Yaskawa INFORM job: KRIS6(-12_90).JBI

/JOB
//NAME KRIS6(-12_90)
//POS
///NPOS 178,178,178,10,0,0
///TOOL 0
///POSTYPE PULSE
///PULSE
C00000=-6764,-164331,-134999,2181,78960,314
C00001=-119255,-47763,-118129,2201,84733,937
C00002=-119348,-33730,-112223,2255,86453,948
C00003=-119057,-93541,-129160,2121,87990,859
C00004=-118979,-101393,-133254,2097,92873,863
C00005=-119932,-77312,-125419,2251,104410,725
C00006=-119932,-79807,-125118,2239,102944,696
C00007=-119932,-78534,-125283,2248,103699,711
C00008=-119946,-74107,-123441,2264,104839,725
C00009=-119932,-78534,-125283,2248,103699,711
C00010=-119867,-91458,-132961,2208,101782,695
C00011=-119929,-73545,-130238,2283,96557,768
C00012=-119929,-73545,-130238,2283,96557,768
C00013=-119957,-58817,-118616,2436,108946,925
C00014=-123171,-49481,-113469,3470,112784,170
C00015=-123153,-49145,-112726,3457,112499,166
C00016=-123153,-51096,-112549,3427,111389,133
C00017=-123153,-49599,-112689,3450,112241,159
C00018=-123109,-46536,-111045,3454,112801,187
C00019=-123280,-52221,-117750,3539,114010,179
C00020=-123574,-64329,-127676,3623,101325,100
C00021=-123574,-64329,-127676,3623,101325,100
C00022=-123766,-59413,-122861,3666,112999,36
C00023=-125942,-52580,-116093,4293,112422,-554
C00024=-126600,-50426,-113316,4465,111850,-748
C00025=-126600,-52772,-113093,4419,110512,-799
C00026=-126600,-51256,-113243,4448,111381,-766
C00027=-126484,-47796,-111410,4439,112022,-709
C00028=-126600,-51256,-113243,4448,111381,-766
C00029=-127517,-71417,-126819,4648,109419,-1089
C00030=-127517,-71417,-126819,4648,95207,-1089
C00031=-127517,-71417,-126819,4648,95207,-1089
C00032=-127517,-73529,-126819,4648,106019,-1089
C00033=-127727,-61749,-119091,4751,107320,-1094
C00034=-130093,-58052,-115859,5494,107341,-1725
C00035=-130093,-60399,-115576,5448,105965,-1787
C00036=-130093,-58676,-115790,5482,106977,-1740
C00037=-129907,-55107,-114011,5451,107705,-1657
C00038=-130162,-58740,-116586,5519,107435,-1737
C00039=-131204,-71916,-126481,5822,106811,-2045
C00040=-131204,-71916,-126481,5822,93687,-2045
C00041=-131204,-71916,-126481,5822,93687,-2045
C00042=-131204,-71916,-126481,5822,105723,-2045
C00043=-130617,-65357,-120996,5631,105686,-1890
C00044=-134640,-60773,-116482,6918,105500,-2981
C00045=-134640,-62624,-116236,6876,104404,-3044
C00046=-134640,-61323,-116413,6905,105177,-2999
C00047=-134343,-57381,-114492,6841,105996,-2874
C00048=-134640,-61323,-116413,6905,105177,-2999
C00049=-133458,-71885,-125928,6541,105529,-2666
C00050=-133867,-78779,-128765,6711,91394,-2865
C00051=-133867,-78779,-128765,6711,91394,-2865
C00052=-133867,-78779,-128765,6711,103158,-2865
C00053=-137702,-64049,-118295,8003,104543,-3826
C00054=-138377,-60786,-116211,8241,104986,-3979
C00055=-138377,-63432,-115832,8173,103411,-4088
C00056=-138377,-61523,-116113,8222,104554,-4010
C00057=-138001,-57618,-114209,8136,105352,-3854
C00058=-138804,-63923,-118462,8370,104797,-4109
C00059=-114789,-54631,-113943,-15836,109322,15159
C00060=-117446,-46661,-107682,-17796,110513,16745
C00061=-135138,-47810,-110215,2755,110872,-639
C00062=-122706,-51038,-111939,2830,110281,-732
C00063=-104898,-47309,-109719,-2181,110784,3733
C00064=-113247,-41947,-106722,9396,112942,-6495
C00065=-115201,-45518,-111139,10036,113978,-6928
C00066=-109888,-67792,-124928,-2208,109623,3796
C00067=-109888,-67792,-124928,-2208,92487,3796
C00068=-109888,-67792,-124928,-2208,92487,3796
C00069=-109888,-67792,-124928,-2208,107991,3796
C00070=-119439,-51982,-113666,11445,111008,-7659
C00071=-117726,-48338,-109777,10887,110325,-7260
C00072=-100866,-50921,-111009,-8782,109155,9371
C00073=-117735,-56763,-114072,-3538,107088,4956
C00074=-137822,-52486,-111893,2748,107867,-389
C00075=-124279,-42666,-106545,-13838,112284,13520
C00076=-119511,-49264,-112664,-15270,113256,14701
C00077=-119402,-57305,-120939,-15547,101345,14582
C00078=-119402,-57305,-120939,-15547,101345,14582
C00079=-119402,-57305,-120939,-15547,109505,14582
C00080=-122292,-51504,-112613,-14389,109095,14125
C00081=-124558,-45323,-107894,-13672,111001,13362
C00082=-143884,-51554,-111193,8957,108316,-5281
C00083=-133478,-57417,-114087,5875,106433,-2802
C00084=-120249,-59696,-115195,2556,105532,-22
C00085=-132290,-46931,-108595,16593,111984,-11759
C00086=-136159,-47694,-113124,18059,114858,-12388
C00087=-139576,-57528,-118771,18775,113901,-13510
C00088=-140360,-69519,-123680,18885,96024,-14170
C00089=-140360,-69519,-123678,18885,96029,-14170
C00090=-141278,-80916,-127529,19144,105606,-14918
C00091=-135966,-58193,-116482,18148,109309,-12780
C00092=-133070,-49776,-109673,17224,110272,-12037
C00093=-115680,-63515,-116432,-2666,103196,4100
C00094=-124283,-63101,-116291,-1790,103261,3381
C00095=-141256,-57210,-113499,5768,104997,-2724
C00096=-125849,-50663,-110250,-12105,107953,11564
C00097=-122691,-57409,-116127,-13110,108460,12368
C00098=-121144,-64717,-120648,-13506,107699,12878
C00099=-121162,-72749,-124196,-13450,93226,13080
C00100=-121162,-72749,-124196,-13450,93226,13080
C00101=-121162,-72749,-124196,-13450,105330,13080
C00102=-121331,-50205,-111480,-16610,110216,14952
C00103=-123990,-47823,-108385,-15715,109173,14365
C00104=-142128,-42054,-107579,5566,113340,-3269
C00105=-131359,-47053,-110363,2420,112110,-462
C00106=-117986,-48725,-111182,-1462,111698,3083
C00107=-133863,-43680,-107086,16750,113488,-14506
C00108=-140868,-51734,-116509,18965,116153,-16042
C00109=-142662,-63919,-124161,19179,114978,-16761
C00110=-142662,-63919,-124161,19179,98114,-16761
C00111=-142662,-63919,-124161,19179,98114,-16761
C00112=-145044,-62011,-123293,19965,112812,-17284
C00113=-140059,-55739,-114817,18192,110093,-16328
C00114=-137449,-52455,-110379,17263,108669,-15828
C00115=-120073,-53031,-112853,-3294,109306,530
C00116=-131848,-51289,-111914,267,109461,-2602
C00117=-144044,-45121,-108584,3992,110813,-5796
C00118=-132169,-40707,-106079,-10221,112829,6404
C00119=-127222,-62973,-118370,-12140,105781,8110
C00120=-127679,-76622,-124397,-11790,102493,8312
C00121=-128554,-105444,-135103,-11820,65639,8862
C00122=-3214,-105444,-135103,-11820,65639,8862
C00123=-61169,66162,-38787,-7489,108505,14459
C00124=-80858,180821,91092,-14176,100483,27377
C00125=-135310,136963,35594,20342,106570,-42107
C00126=-129648,130678,34027,17726,103545,-41191
C00127=-129561,130561,33941,17673,103533,-41171
C00128=-129561,128436,32943,17631,103075,-41240
C00129=-129561,129425,33401,17649,103291,-41208
C00130=-128781,129160,33005,17330,103280,-41016
C00131=-129561,130132,33735,17661,103442,-41185
C00132=-139750,134137,8010,38577,113267,-40747
C00133=-139750,125190,2929,38142,112100,-41205
C00134=-139699,124063,2750,37981,111721,-41340
C00135=-139750,125190,2929,38142,112100,-41205
C00136=-139020,124881,2398,37778,112092,-41058
C00137=-139750,125190,2929,38142,112100,-41205
C00138=-139750,125190,2929,38142,112100,-41205
C00139=-106399,146658,29541,9597,114270,-2674
C00140=-80858,180821,91092,-14176,100483,27377
C00141=-112418,209939,108052,-33593,108566,52711
C00142=-113977,200131,96183,-33565,110017,51753
C00143=-113977,196712,92480,-33687,110454,51613
C00144=-113977,198404,94297,-33628,110245,51681
C00145=-114566,198013,93705,-33460,110217,51508
C00146=-112711,202956,96769,-34269,111286,51731
C00147=-115091,169447,47419,-27866,117108,43490
C00148=-116360,163418,42413,-27282,116877,43269
C00149=-116606,162287,41507,-27163,116815,43231
C00150=-116612,160850,40689,-27099,116604,43286
C00151=-116606,162287,41507,-27163,116815,43231
C00152=-117158,162218,41388,-26920,116756,43124
C00153=-115998,165435,44045,-27455,116968,43326
C00154=-112418,209939,108052,-33593,108566,52711
C00155=-114652,201087,99032,-33053,108767,51943
C00156=-114651,200952,98830,-33066,108814,51929
C00157=-114319,178188,64429,-35758,116797,49311
C00158=-117155,160465,40052,-26903,116688,43142
C00159=-116538,119181,-10894,-26822,112395,43970
C00160=-116367,70767,-36778,-25412,104337,45903
C00161=-114627,81723,-35948,-27198,109202,45070
C00162=-114627,81723,-35948,-27198,109202,45070
C00163=-115397,82628,-35755,-25618,94251,45537
C00164=-143127,87221,-28738,37921,95336,-39907
C00165=-140662,151607,34414,42484,118899,-37225
C00166=-138525,189832,83608,37500,122713,-39265
C00167=-136744,206891,106864,34388,120949,-40419
C00168=-136748,206624,106472,34429,121037,-40387
C00169=-137297,183579,72826,37483,123882,-38878
C00170=-137988,166130,49785,38283,120093,-39568
C00171=-139920,130462,7613,39720,110784,-41477
C00172=-141169,114879,-10138,41320,113277,-40682
C00173=-142291,101361,-22992,42309,114215,-40480
C00174=-127329,75853,-46961,19716,114528,-24997
C00175=-127329,75853,-46961,19716,114528,-24997
C00176=-19661,75853,-46961,19716,114528,-24997
C00177=-3214,-105444,-135103,-11820,65639,8862
BC00000=123481,666391,1059275
BC00001=123481,666391,1059275
BC00002=68091,722952,1059275
BC00003=68091,757345,1059275
BC00004=71245,776429,1059275
BC00005=71244,776429,1059274
BC00006=71244,776429,1059274
BC00007=71244,776429,1059274
BC00008=71244,776429,1059274
BC00009=71244,776429,1059274
BC00010=71244,776429,1059274
BC00011=71244,750340,1059274
BC00012=148732,750340,1059274
BC00013=148732,764150,1059274
BC00014=148732,764150,1059274
BC00015=148732,764150,1059274
BC00016=148732,764150,1059274
BC00017=148732,764150,1059274
BC00018=148732,764150,1059274
BC00019=148732,764150,1059274
BC00020=148732,764150,1059274
BC00021=205656,764150,1059274
BC00022=205656,764150,1059274
BC00023=205656,764150,1059274
BC00024=205656,764150,1059274
BC00025=205656,764150,1059274
BC00026=205656,764150,1059274
BC00027=205656,764150,1059274
BC00028=205656,764150,1059274
BC00029=205656,764150,1059274
BC00030=205656,764150,1059274
BC00031=262390,764150,1059274
BC00032=262390,764150,1059274
BC00033=262390,764150,1059274
BC00034=262390,764150,1059274
BC00035=262390,764150,1059274
BC00036=262390,764150,1059274
BC00037=262390,764150,1059274
BC00038=262390,764150,1059274
BC00039=262390,764150,1059274
BC00040=262390,764150,1059274
BC00041=297084,764150,1059274
BC00042=297084,764150,1059274
BC00043=297084,764150,1059274
BC00044=297084,764150,1059274
BC00045=297084,764150,1059274
BC00046=297084,764150,1059274
BC00047=297084,764150,1059274
BC00048=297084,764150,1059274
BC00049=297084,764150,1059274
BC00050=297084,764150,1059274
BC00051=377314,764150,1059274
BC00052=377314,764150,1059274
BC00053=377314,764150,1059274
BC00054=377314,764150,1059274
BC00055=377314,764150,1059274
BC00056=377314,764150,1059274
BC00057=377314,764150,1059274
BC00058=377314,764150,1059274
BC00059=345104,764150,1059274
BC00060=345104,764150,1059271
BC00061=345104,764150,1059271
BC00062=345104,764150,1059271
BC00063=345104,764149,1059267
BC00064=345104,764149,1059267
BC00065=345104,764149,1059267
BC00066=345104,764149,1059267
BC00067=345104,764149,1059267
BC00068=92083,764149,1059267
BC00069=92083,764149,1059267
BC00070=92084,764149,1059264
BC00071=92084,764149,1059261
BC00072=92084,764149,1059261
BC00073=92084,764149,1059261
BC00074=92084,764149,1059261
BC00075=92084,764149,1059261
BC00076=92084,764149,1059261
BC00077=92084,764149,1059261
BC00078=208313,764149,1059261
BC00079=208313,764149,1059261
BC00080=208313,764149,1059257
BC00081=208313,764149,1059257
BC00082=208313,764149,1059257
BC00083=208313,764149,1059257
BC00084=208313,764149,1059254
BC00085=208313,764149,1059254
BC00086=208313,764149,1059254
BC00087=208313,764149,1059254
BC00088=208313,764149,1059254
BC00089=304618,764149,1059250
BC00090=304618,764149,1059250
BC00091=304618,764149,1059250
BC00092=304618,764149,1059250
BC00093=304618,764149,1059250
BC00094=304618,764149,1059250
BC00095=304618,764149,1059250
BC00096=304619,764149,1059247
BC00097=304619,764149,1059247
BC00098=304619,764149,1059247
BC00099=304619,764149,1059247
BC00100=163196,764149,1059247
BC00101=163196,764149,1059247
BC00102=163195,764149,1059243
BC00103=163195,764149,1059243
BC00104=163195,764149,1059243
BC00105=163195,764149,1059243
BC00106=163195,764149,1059243
BC00107=163195,764149,1059243
BC00108=163195,764149,1059243
BC00109=163195,764149,1059243
BC00110=163195,764149,1059243
BC00111=264866,764149,1059243
BC00112=264866,764149,1059243
BC00113=264866,764149,1059243
BC00114=264866,764149,1059243
BC00115=264866,764149,1059243
BC00116=264866,764149,1059243
BC00117=264866,764149,1059243
BC00118=264866,764149,1059243
BC00119=264866,764149,1059243
BC00120=264866,764149,1059243
BC00121=264866,753228,1059243
BC00122=191713,674662,1052383
BC00123=157008,682575,1029984
BC00124=131441,688404,1013483
BC00125=377113,693279,1026468
BC00126=377113,693279,1026468
BC00127=377112,693278,1026465
BC00128=377112,693278,1026465
BC00129=377112,693278,1026465
BC00130=377112,693278,1026465
BC00131=377112,693278,1026465
BC00132=383615,696698,828304
BC00133=383615,696698,828304
BC00134=383614,696697,828301
BC00135=383615,696698,828304
BC00136=383615,696698,828304
BC00137=383615,696698,828304
BC00138=376930,696698,899272
BC00139=245359,692151,929829
BC00140=131441,688404,1013483
BC00141=92845,712939,790660
BC00142=92845,712939,790660
BC00143=92845,712939,790660
BC00144=92845,712939,790660
BC00145=92845,712939,790660
BC00146=92845,712939,790660
BC00147=92845,693279,790660
BC00148=92845,693279,790660
BC00149=92845,693279,790660
BC00150=92845,693279,790660
BC00151=92845,693279,790660
BC00152=92845,693279,790660
BC00153=92845,693279,790660
BC00154=92845,712939,790660
BC00155=92845,712939,790660
BC00156=92845,712939,790660
BC00157=92845,712939,790660
BC00158=92845,693279,790660
BC00159=92845,693279,790660
BC00160=92845,693279,946108
BC00161=92845,693279,946108
BC00162=377113,693279,946108
BC00163=377113,693279,1026468
BC00164=377113,693279,1026468
BC00165=381773,721654,941888
BC00166=383883,734501,832605
BC00167=384437,737875,803900
BC00168=384437,737875,803900
BC00169=384437,727595,803897
BC00170=384437,710229,803249
BC00171=384437,697061,803249
BC00172=384437,697061,803249
BC00173=384437,697061,803249
BC00174=345074,693590,934356
BC00175=345074,674682,934356
BC00176=207964,677290,934356
BC00177=191713,674662,1052383
EC00000=-106353,556476
EC00001=-106353,556476
EC00002=-106353,556476
EC00003=-106353,556476
EC00004=-106353,556476
EC00005=-106351,556476
EC00006=-106351,556476
EC00007=-106351,556476
EC00008=-106351,556476
EC00009=-106351,556476
EC00010=-106351,556476
EC00011=-106351,556476
EC00012=-106351,556476
EC00013=-106351,556476
EC00014=-106351,556476
EC00015=-106351,556476
EC00016=-106351,556476
EC00017=-106351,556476
EC00018=-106351,556476
EC00019=-106351,556476
EC00020=-106351,556476
EC00021=-106351,556476
EC00022=-106351,556476
EC00023=-106351,556476
EC00024=-106351,556476
EC00025=-106351,556476
EC00026=-106351,556476
EC00027=-106351,556476
EC00028=-106351,556476
EC00029=-106351,556476
EC00030=-106351,556476
EC00031=-106351,556476
EC00032=-106351,556476
EC00033=-106351,556476
EC00034=-106351,556476
EC00035=-106351,556476
EC00036=-106351,556476
EC00037=-106351,556476
EC00038=-106351,556476
EC00039=-106351,556476
EC00040=-106351,556476
EC00041=-106351,556476
EC00042=-106351,556476
EC00043=-106351,556476
EC00044=-106351,556476
EC00045=-106351,556476
EC00046=-106351,556476
EC00047=-106351,556476
EC00048=-106351,556476
EC00049=-106351,556476
EC00050=-106351,556476
EC00051=-106351,556476
EC00052=-106351,556476
EC00053=-106351,556476
EC00054=-106351,556476
EC00055=-106351,556476
EC00056=-106351,556476
EC00057=-106351,556476
EC00058=-106351,556476
EC00059=-106351,556476
EC00060=-106350,556477
EC00061=-106350,556477
EC00062=-106350,556477
EC00063=-106350,556477
EC00064=-106350,556477
EC00065=-106350,556477
EC00066=-106350,556477
EC00067=-106350,556477
EC00068=-106350,556477
EC00069=-106350,556477
EC00070=-106349,556477
EC00071=-106348,556477
EC00072=-106348,556477
EC00073=-106348,556477
EC00074=-106348,556477
EC00075=-106348,556477
EC00076=-106348,556477
EC00077=-106348,556477
EC00078=-106348,556477
EC00079=-106348,556477
EC00080=-106348,556477
EC00081=-106348,556477
EC00082=-106348,556477
EC00083=-106348,556477
EC00084=-106347,556477
EC00085=-106347,556477
EC00086=-106347,556477
EC00087=-106347,556477
EC00088=-106347,556477
EC00089=-106347,556477
EC00090=-106347,556477
EC00091=-106347,556477
EC00092=-106347,556477
EC00093=-106347,556477
EC00094=-106347,556477
EC00095=-106347,556477
EC00096=-106346,556477
EC00097=-106346,556477
EC00098=-106346,556477
EC00099=-106346,556477
EC00100=-106346,556477
EC00101=-106346,556477
EC00102=-106346,556477
EC00103=-106346,556477
EC00104=-106346,556477
EC00105=-106346,556477
EC00106=-106346,556477
EC00107=-106346,556477
EC00108=-106346,556477
EC00109=-106346,556477
EC00110=-106346,556477
EC00111=-106346,556477
EC00112=-106346,556477
EC00113=-106346,556477
EC00114=-106346,556477
EC00115=-106346,556477
EC00116=-106346,556477
EC00117=-106346,556477
EC00118=-106346,556477
EC00119=-106346,556477
EC00120=-106346,556477
EC00121=-106346,556477
EC00122=-106346,556477
EC00123=-307585,556477
EC00124=-455838,556477
EC00125=-458173,556477
EC00126=-458173,556477
EC00127=-458170,556478
EC00128=-458170,556478
EC00129=-458170,556478
EC00130=-458170,556478
EC00131=-458170,556478
EC00132=-458171,556477
EC00133=-458171,556477
EC00134=-458169,556477
EC00135=-458171,556477
EC00136=-458171,556477
EC00137=-458171,556477
EC00138=-458171,556477
EC00139=-456892,556477
EC00140=-455838,556477
EC00141=-458173,556477
EC00142=-458173,556477
EC00143=-458173,556477
EC00144=-458173,556477
EC00145=-458173,556477
EC00146=-458173,556477
EC00147=-458173,556477
EC00148=-458173,556477
EC00149=-458173,556477
EC00150=-458173,556477
EC00151=-458173,556477
EC00152=-458173,556477
EC00153=-458173,556477
EC00154=-458173,556477
EC00155=-458173,556477
EC00156=-458173,556477
EC00157=-458173,556477
EC00158=-458173,556477
EC00159=-458173,556477
EC00160=-458173,556477
EC00161=-458173,556477
EC00162=-458173,556477
EC00163=-458173,556477
EC00164=-458173,556477
EC00165=-458173,556477
EC00166=-458173,556477
EC00167=-458173,556477
EC00168=-458173,556477
EC00169=-458171,556477
EC00170=-458171,556477
EC00171=-458171,556477
EC00172=-458171,556477
EC00173=-458171,556477
EC00174=-458173,556477
EC00175=-458173,556477
EC00176=-458173,556477
EC00177=-106346,556477
///POSTYPE BASE
///RECTAN
///RCONF 0,0,0,0,0,0,0,0,0,0,0,0,0,0,0,0,0,0,0,0,0,0,0,0
P00006=0.222,-3.123,-1.508,0.0000,0.0000,0.0000
P00021=-0.225,-6.128,-0.405,0.0000,0.0000,0.0000
P00022=0.222,-3.123,-1.508,0.0000,0.0000,0.0000
P00023=0.143,-0.036,0.682,0.0000,0.0000,0.0000
P00024=0.145,-0.552,1.326,0.0000,0.0000,0.0000
P00025=-2.003,0.006,0.728,0.0000,0.0000,0.0000
P00026=0.562,-0.002,-0.337,0.0000,0.0000,0.0000
P00027=-0.746,0.015,-9.096,0.0000,0.0000,0.0000
P00028=-2.237,-0.018,-7.702,0.0000,0.0000,0.0000
P00029=-2.156,-0.086,-4.681,0.0000,0.0000,0.0000
//INST
///DATE 2025/01/14 08:36
///COMM SPOINY POMIEDZY ZEBRAMI
///ATTR SC,RW
///GROUP1 RB1,BS1
///GROUP2 ST1
NOP
'MUZYLO 310124 PISANIE NOWEGO PRO
MOVJ C00000 BC00000 VJ=100.00  +MOVJ EC00000 VJ=100.00
MOVJ C00001 BC00001 VJ=100.00  +MOVJ EC00001 VJ=100.00
MOVJ C00002 BC00002 VJ=100.00  +MOVJ EC00002 VJ=100.00
MOVJ C00003 BC00003 VJ=100.00  +MOVJ EC00003 VJ=100.00
MOVJ C00004 BC00004 VJ=100.00  +MOVJ EC00004 VJ=100.00
SMOVL C00005 BC00005 V=100.0  +MOVJ EC00005
SREFP 3 C00006 BC00006  +REFP EC00006
CALL JOB:SEARCH-R1-S13D
SET P021 P006
SFTON3D P021
SMOVL C00007 BC00007 V=100.0  +MOVJ EC00007
SREFP 3 C00008 BC00008  +REFP EC00008
CALL JOB:SEARCH-R1-S13D
SET P021 P006
SMOVL C00009 BC00009 V=133.3  +MOVJ EC00009
SFTOF3D
MOVJ C00010 BC00010 VJ=100.00  +MOVJ EC00010 VJ=100.00
MOVJ C00011 BC00011 VJ=100.00  +MOVJ EC00011 VJ=100.00
MOVJ C00012 BC00012 VJ=100.00  +MOVJ EC00012 VJ=100.00
MOVJ C00013 BC00013 VJ=100.00  +MOVJ EC00013 VJ=100.00
MOVJ C00014 BC00014 VJ=100.00  +MOVJ EC00014 VJ=100.00
SMOVL C00015 BC00015 V=100.0  +MOVJ EC00015
SREFP 3 C00016 BC00016  +REFP EC00016
CALL JOB:SEARCH-R1-S13D
SET P022 P006
SFTON3D P022
SMOVL C00017 BC00017 V=100.0  +MOVJ EC00017
SREFP 3 C00018 BC00018  +REFP EC00018
CALL JOB:SEARCH-R1-S13D
SET P022 P006
SFTON3D P022
SFTOF3D
SMOVL C00019 BC00019 V=166.7  +MOVJ EC00019
MOVJ C00020 BC00020 VJ=100.00  +MOVJ EC00020 VJ=100.00
MOVJ C00021 BC00021 VJ=100.00  +MOVJ EC00021 VJ=100.00
MOVJ C00022 BC00022 VJ=100.00  +MOVJ EC00022 VJ=100.00
MOVJ C00023 BC00023 VJ=100.00  +MOVJ EC00023 VJ=100.00
SMOVL C00024 BC00024 V=100.0  +MOVJ EC00024
SREFP 3 C00025 BC00025  +REFP EC00025
CALL JOB:SEARCH-R1-S13D
SET P023 P006
SFTON3D P023
SMOVL C00026 BC00026 V=100.0  +MOVJ EC00026
SREFP 3 C00027 BC00027  +REFP EC00027
CALL JOB:SEARCH-R1-S13D
SET P023 P006
SFTON3D P023
SFTOF3D
SMOVL C00028 BC00028 V=133.3  +MOVJ EC00028
MOVJ C00029 BC00029 VJ=100.00  +MOVJ EC00029 VJ=100.00
MOVJ C00030 BC00030 VJ=100.00  +MOVJ EC00030 VJ=100.00
MOVJ C00031 BC00031 VJ=100.00  +MOVJ EC00031 VJ=100.00
MOVJ C00032 BC00032 VJ=100.00  +MOVJ EC00032 VJ=100.00
MOVJ C00033 BC00033 VJ=100.00  +MOVJ EC00033 VJ=100.00
SMOVL C00034 BC00034 V=100.0  +MOVJ EC00034
SREFP 3 C00035 BC00035  +REFP EC00035
CALL JOB:SEARCH-R1-S13D
SET P024 P006
SFTON3D P024
SMOVL C00036 BC00036 V=100.0  +MOVJ EC00036
SREFP 3 C00037 BC00037  +REFP EC00037
CALL JOB:SEARCH-R1-S13D
SET P024 P006
SFTON3D P024
SFTOF3D
SMOVL C00038 BC00038 V=166.7  +MOVJ EC00038
MOVJ C00039 BC00039 VJ=100.00  +MOVJ EC00039 VJ=100.00
MOVJ C00040 BC00040 VJ=100.00  +MOVJ EC00040 VJ=100.00
MOVJ C00041 BC00041 VJ=100.00  +MOVJ EC00041 VJ=100.00
MOVJ C00042 BC00042 VJ=100.00  +MOVJ EC00042 VJ=100.00
MOVJ C00043 BC00043 VJ=100.00  +MOVJ EC00043 VJ=100.00
SMOVL C00044 BC00044 V=100.0  +MOVJ EC00044
SREFP 3 C00045 BC00045  +REFP EC00045
CALL JOB:SEARCH-R1-S13D
SET P025 P006
SFTON3D P025
SMOVL C00046 BC00046 V=100.0  +MOVJ EC00046
SREFP 3 C00047 BC00047  +REFP EC00047
CALL JOB:SEARCH-R1-S13D
SET P025 P006
SFTON3D P025
SFTOF3D
SMOVL C00048 BC00048 V=166.7  +MOVJ EC00048
MOVJ C00049 BC00049 VJ=100.00  +MOVJ EC00049 VJ=100.00
MOVJ C00050 BC00050 VJ=100.00  +MOVJ EC00050 VJ=100.00
MOVJ C00051 BC00051 VJ=100.00  +MOVJ EC00051 VJ=100.00
MOVJ C00052 BC00052 VJ=100.00  +MOVJ EC00052 VJ=100.00
MOVJ C00053 BC00053 VJ=100.00  +MOVJ EC00053 VJ=100.00
SMOVL C00054 BC00054 V=100.0  +MOVJ EC00054
SREFP 3 C00055 BC00055  +REFP EC00055
CALL JOB:SEARCH-R1-S13D
SET P026 P006
SFTON3D P026
SMOVL C00056 BC00056 V=100.0  +MOVJ EC00056
SREFP 3 C00057 BC00057  +REFP EC00057
CALL JOB:SEARCH-R1-S13D
SET P026 P006
SMOVL C00058 BC00058 V=166.7  +MOVJ EC00058
MOVJ C00059 BC00059 VJ=100.00  +MOVJ EC00059 VJ=100.00
MACRO1 MJ#(0) ARGF9
SFTON3D P026
SMOVL C00060 BC00060 V=133.3  +MOVJ EC00060
ARCON
SMOVL C00061 BC00061 V=8.3  +MOVJ EC00061
SMOVL C00062 BC00062 V=8.3  +MOVJ EC00062
SMOVL C00063 BC00063 V=8.3  +MOVJ EC00063
SMOVL C00064 BC00064 V=8.3  +MOVJ EC00064
ARCOF
SFTOF3D
SMOVL C00065 BC00065 V=166.7  +MOVJ EC00065
MOVJ C00066 BC00066 VJ=100.00  +MOVJ EC00066 VJ=100.00
MOVJ C00067 BC00067 VJ=100.00  +MOVJ EC00067 VJ=100.00
MOVJ C00068 BC00068 VJ=100.00  +MOVJ EC00068 VJ=100.00
MOVJ C00069 BC00069 VJ=100.00  +MOVJ EC00069 VJ=100.00
MOVJ C00070 BC00070 VJ=100.00  +MOVJ EC00070 VJ=100.00
SFTON3D P021
SMOVL C00071 BC00071 V=133.3  +MOVJ EC00071
ARCON
SMOVL C00072 BC00072 V=8.3  +MOVJ EC00072
SMOVL C00073 BC00073 V=8.3  +MOVJ EC00073
SMOVL C00074 BC00074 V=8.3  +MOVJ EC00074
SMOVL C00075 BC00075 V=8.3  +MOVJ EC00075
ARCOF
SFTOF3D
MOVJ C00076 BC00076 VJ=100.00  +MOVJ EC00076 VJ=100.00
MOVJ C00077 BC00077 VJ=100.00  +MOVJ EC00077 VJ=100.00
MOVJ C00078 BC00078 VJ=100.00  +MOVJ EC00078 VJ=100.00
MOVJ C00079 BC00079 VJ=100.00  +MOVJ EC00079 VJ=100.00
MOVJ C00080 BC00080 VJ=100.00  +MOVJ EC00080 VJ=100.00
SFTON3D P023
SMOVL C00081 BC00081 V=133.3  +MOVJ EC00081
ARCON
SMOVL C00082 BC00082 V=8.3  +MOVJ EC00082
SMOVL C00083 BC00083 V=8.3  +MOVJ EC00083
SMOVL C00084 BC00084 V=8.3  +MOVJ EC00084
SMOVL C00085 BC00085 V=8.3  +MOVJ EC00085
ARCOF
SFTOF3D
SMOVL C00086 BC00086 V=166.7  +MOVJ EC00086
MOVJ C00087 BC00087 VJ=100.00  +MOVJ EC00087 VJ=100.00
MOVJ C00088 BC00088 VJ=100.00  +MOVJ EC00088 VJ=100.00
MOVJ C00089 BC00089 VJ=100.00  +MOVJ EC00089 VJ=100.00
MOVJ C00090 BC00090 VJ=100.00  +MOVJ EC00090 VJ=100.00
MOVJ C00091 BC00091 VJ=100.00  +MOVJ EC00091 VJ=100.00
SFTON3D P025
SMOVL C00092 BC00092 V=133.3  +MOVJ EC00092
ARCON
SMOVL C00093 BC00093 V=8.3  +MOVJ EC00093
SMOVL C00094 BC00094 V=8.3  +MOVJ EC00094
SMOVL C00095 BC00095 V=8.3  +MOVJ EC00095
SMOVL C00096 BC00096 V=8.3  +MOVJ EC00096
ARCOF
SFTOF3D
SMOVL C00097 BC00097 V=133.3  +MOVJ EC00097
MOVJ C00098 BC00098 VJ=100.00  +MOVJ EC00098 VJ=100.00
MOVJ C00099 BC00099 VJ=100.00  +MOVJ EC00099 VJ=100.00
MOVJ C00100 BC00100 VJ=100.00  +MOVJ EC00100 VJ=100.00
MOVJ C00101 BC00101 VJ=100.00  +MOVJ EC00101 VJ=100.00
MOVJ C00102 BC00102 VJ=100.00  +MOVJ EC00102 VJ=100.00
SFTON3D P022
SMOVL C00103 BC00103 V=133.3  +MOVJ EC00103
ARCON
SMOVL C00104 BC00104 V=7.5  +MOVJ EC00104
SMOVL C00105 BC00105 V=7.5  +MOVJ EC00105
SMOVL C00106 BC00106 V=7.5  +MOVJ EC00106
SMOVL C00107 BC00107 V=7.5  +MOVJ EC00107
ARCOF
SFTOF3D
SMOVL C00108 BC00108 V=166.7  +MOVJ EC00108
MOVJ C00109 BC00109 VJ=100.00  +MOVJ EC00109 VJ=100.00
MOVJ C00110 BC00110 VJ=100.00  +MOVJ EC00110 VJ=100.00
MOVJ C00111 BC00111 VJ=100.00  +MOVJ EC00111 VJ=100.00
MOVJ C00112 BC00112 VJ=100.00  +MOVJ EC00112 VJ=100.00
MOVJ C00113 BC00113 VJ=100.00  +MOVJ EC00113 VJ=100.00
SFTON3D P024
SMOVL C00114 BC00114 V=133.3  +MOVJ EC00114
ARCON
SMOVL C00115 BC00115 V=7.5  +MOVJ EC00115
SMOVL C00116 BC00116 V=7.5  +MOVJ EC00116
SMOVL C00117 BC00117 V=7.5  +MOVJ EC00117
SMOVL C00118 BC00118 V=7.5  +MOVJ EC00118
ARCOF
SFTOF3D
SMOVL C00119 BC00119 V=166.7  +MOVJ EC00119
MOVJ C00120 BC00120 VJ=100.00  +MOVJ EC00120 VJ=100.00
MOVJ C00121 BC00121 VJ=100.00  +MOVJ EC00121 VJ=100.00
MOVJ C00122 BC00122 VJ=100.00  +MOVJ EC00122 VJ=100.00
CALL JOB:CLEAN-R1_KM_3P
'MAX DO -52ST
MOVJ C00123 BC00123 VJ=100.00  +MOVJ EC00123 VJ=100.00
SFTOF3D
SFTOF3D
SFTOF
MOVJ C00124 BC00124 VJ=100.00  +MOVJ EC00124 VJ=100.00
MOVJ C00125 BC00125 VJ=100.00  +MOVJ EC00125 VJ=100.00
MOVJ C00126 BC00126 VJ=100.00  +MOVJ EC00126 VJ=100.00
'SEARCH-1
SMOVL C00127 BC00127 V=100.0  +MOVJ EC00127
SREFP 3 C00128 BC00128  +REFP EC00128
CALL JOB:SEARCH-R1-S13D
SET P026 P006
SFTON3D P026
SMOVL C00129 BC00129 V=100.0  +MOVJ EC00129
SREFP 3 C00130 BC00130  +REFP EC00130
CALL JOB:SEARCH-R1-S13D
SET P026 P006
SFTON3D P026
SFTOF3D
SMOVL C00131 BC00131 V=166.7  +MOVJ EC00131
SFTOF3D
SMOVL C00132 BC00132 V=333.3  +MOVJ EC00132
SMOVL C00133 BC00133 V=100.0  +MOVJ EC00133
SREFP 3 C00134 BC00134  +REFP EC00134
CALL JOB:SEARCH-R1-S13D
SET P028 P006
SFTON3D P028
SMOVL C00135 BC00135 V=100.0  +MOVJ EC00135
SREFP 3 C00136 BC00136  +REFP EC00136
CALL JOB:SEARCH-R1-S13D
SET P028 P006
SFTON3D P028
SFTOF3D
SMOVL C00137 BC00137 V=166.7  +MOVJ EC00137
MOVJ C00138 BC00138 VJ=70.00  +MOVJ EC00138 VJ=70.00
SFTOF3D
MOVJ C00139 BC00139 VJ=70.00  +MOVJ EC00139 VJ=70.00
MOVJ C00140 BC00140 VJ=100.00  +MOVJ EC00140 VJ=10.00
MOVJ C00141 BC00141 VJ=100.00  +MOVJ EC00141 VJ=50.00
'SEARCH-2
SMOVL C00142 BC00142 V=100.0  +MOVJ EC00142
SREFP 3 C00143 BC00143  +REFP EC00143
CALL JOB:SEARCH-R1-S13D
SET P027 P006
SFTON3D P027
SMOVL C00144 BC00144 V=100.0  +MOVJ EC00144
SREFP 3 C00145 BC00145  +REFP EC00145
CALL JOB:SEARCH-R1-S13D
SET P027 P006
SFTON3D P027
SMOVL C00146 BC00146 V=250.0  +MOVJ EC00146
SFTOF3D
MOVJ C00147 BC00147 VJ=70.00  +MOVJ EC00147 VJ=70.00
MOVJ C00148 BC00148 VJ=70.00  +MOVJ EC00148 VJ=70.00
SMOVL C00149 BC00149 V=100.0  +MOVJ EC00149
SREFP 3 C00150 BC00150  +REFP EC00150
CALL JOB:SEARCH-R1-S13D
SET P029 P006
SFTON3D P029
SMOVL C00151 BC00151 V=100.0  +MOVJ EC00151
SREFP 3 C00152 BC00152  +REFP EC00152
CALL JOB:SEARCH-R1-S13D
SET P029 P006
SFTON3D P029
SFTOF3D
SMOVL C00153 BC00153 V=166.7  +MOVJ EC00153
MOVJ C00154 BC00154 VJ=100.00  +MOVJ EC00154 VJ=100.00
MACRO1 MJ#(0) ARGF21
SFTON3D P027
SMOVL C00155 BC00155 V=133.3  +MOVJ EC00155
ARCON
SMOVC C00156 BC00156 V=10.0  +MOVJ EC00156
SMOVC C00157 BC00157 V=10.0  +MOVJ EC00157
SFTON3D P029
SMOVC C00158 BC00158 V=10.0  +MOVJ EC00158
SMOVC C00159 BC00159 V=10.0  +MOVJ EC00159
SMOVC C00160 BC00160 V=10.0  +MOVJ EC00160
ARCOF
SFTOF3D
SMOVL C00161 BC00161 V=166.7  +MOVJ EC00161
SMOVL C00162 BC00162 V=1000.0  +MOVJ EC00162
MOVJ C00163 BC00163 VJ=100.00  +MOVJ EC00163 VJ=100.00
MOVJ C00164 BC00164 VJ=100.00  +MOVJ EC00164 VJ=100.00
MOVJ C00165 BC00165 VJ=100.00  +MOVJ EC00165 VJ=10.00
SMOVL C00166 BC00166 V=500.0  +MOVJ EC00166
SFTON3D P026
SMOVL C00167 BC00167 V=166.7  +MOVJ EC00167
ARCON
SMOVC C00168 BC00168 V=10.0  +MOVJ EC00168
SMOVC C00169 BC00169 V=10.0  +MOVJ EC00169
SMOVC C00170 BC00170 V=10.0  +MOVJ EC00170
SFTON3D P028
SMOVC C00171 BC00171 V=10.0  +MOVJ EC00171
SMOVC C00172 BC00172 V=10.0  +MOVJ EC00172
SMOVC C00173 BC00173 V=10.0  +MOVJ EC00173
ARCOF
SFTOF3D
SMOVL C00174 BC00174 V=166.7  +MOVJ EC00174
MOVJ C00175 BC00175 VJ=100.00  +MOVJ EC00175 VJ=100.00
MOVJ C00176 BC00176 VJ=100.00  +MOVJ EC00176 VJ=100.00
MOVJ C00177 BC00177 VJ=100.00  +MOVJ EC00177 VJ=100.00
END
